// LS Electric XG5000 project: 71회예상2_2
// PLC NewPLC
// module base 0 slot 0: 입출력 모듈:XBC-DR20S (DC 24V 입력 12점, 릴레이 출력 8점)

PROGRAM NewProgram (task: 스캔 프로그램)

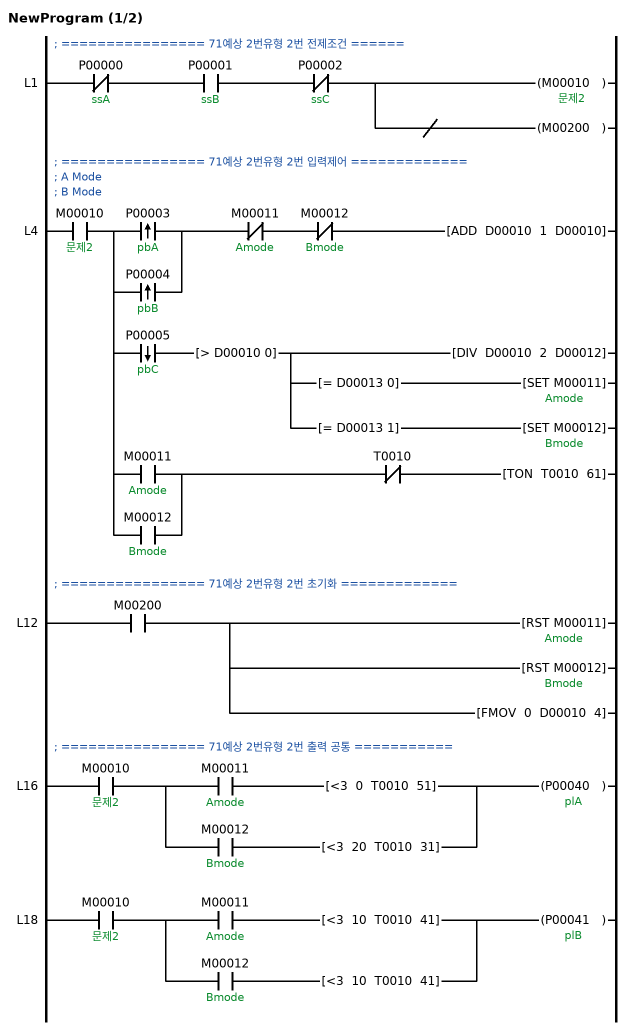
// ================ 71예상 2번유형 2번 전제조건 ======
; L1
LOAD NOT  P00000	// ssA
AND       P00001	// ssB
AND NOT   P00002	// ssC
OUT       M00010	// 문제2
NOT
OUT       M00200
// ================ 71예상 2번유형 2번 입력제어 =============
; L4
LOAD      M00010	// 문제2
MPUSH
LOADP     P00003	// pbA
ORP       P00004	// pbB
AND LOAD
AND NOT   M00011	// Amode
AND NOT   M00012	// Bmode
ADD       D00010 1 D00010
MLOAD
ANDN      P00005	// pbC
AND>      D00010 0
DIV       D00010 2 D00012
MPUSH
AND=      D00013 0
SET       M00011	// Amode
MPOP
AND=      D00013 1
SET       M00012	// Bmode
MPOP
LOAD      M00011	// Amode
OR        M00012	// Bmode
AND LOAD
AND NOT   T0010
TON       T0010 61
// output comment: A Mode
// output comment: B Mode
// ================ 71예상 2번유형 2번 초기화 =============
; L12
LOAD      M00200
RST       M00011	// Amode
RST       M00012	// Bmode
FMOV      0 D00010 4
// ================ 71예상 2번유형 2번 출력 공통 ===========
; L16
LOAD      M00010	// 문제2
LOAD      M00011	// Amode
AND<3     0 T0010 51
LOAD      M00012	// Bmode
AND<3     20 T0010 31
OR LOAD
AND LOAD
OUT       P00040	// plA
; L18
LOAD      M00010	// 문제2
LOAD      M00011	// Amode
AND<3     10 T0010 41
LOAD      M00012	// Bmode
AND<3     10 T0010 41
OR LOAD
AND LOAD
OUT       P00041	// plB

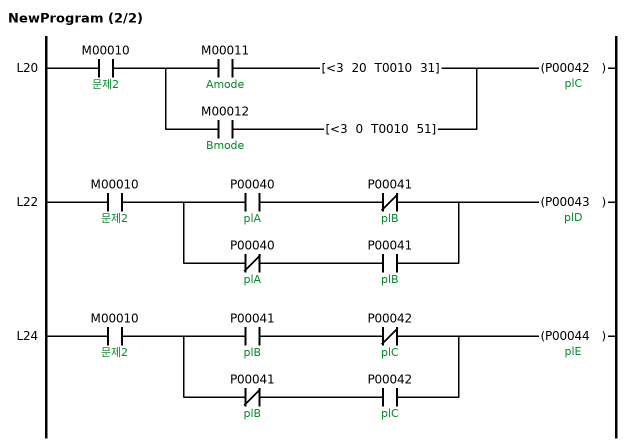
; L20
LOAD      M00010	// 문제2
LOAD      M00011	// Amode
AND<3     20 T0010 31
LOAD      M00012	// Bmode
AND<3     0 T0010 51
OR LOAD
AND LOAD
OUT       P00042	// plC
; L22
LOAD      M00010	// 문제2
LOAD      P00040	// plA
AND NOT   P00041	// plB
LOAD NOT  P00040	// plA
AND       P00041	// plB
OR LOAD
AND LOAD
OUT       P00043	// plD
; L24
LOAD      M00010	// 문제2
LOAD      P00041	// plB
AND NOT   P00042	// plC
LOAD NOT  P00041	// plB
AND       P00042	// plC
OR LOAD
AND LOAD
OUT       P00044	// plE